FUNCTION_BLOCK TimeChannel1CH
VAR_INPUT
	EN: BOOL := TRUE;// Enable the time channel (settings must also be enabled)
	Speed            : INT;		// $(skip) 0,1=normal speed, 2=high speed
	OnTime           : UINT;	(* Hour/minute value of the switch-on time on the day *)
	OffTime          : UINT := 2400;	(* Hour/minute value of the switch-off time on the day *)
	Day: TimerDays;
	SingleShot       : BOOL;	(* $(skip) Resets EN after the on/off cycle is complete *)   
END_VAR
VAR_OUTPUT
	ENO: BOOL; // $(skip) Set if enabled and settings are valid
	Q: BOOL; // Result of the time channel
	Error: BOOL; // Settings error
	ErrorID: UDINT; // // $(skip) 1 = Inconsistent weekday settings, 2 = Bad time settings, 3 = on and off times equal
END_VAR
VAR
	CurrentDay: WORD; // $(skip)
	DayMatch: BOOL; // $(skip)
	LocalSystemTime: FB_LocalSystemTime; // $(skip)
	IsOnTime: BOOL; // $(skip)
	MinuteOfDay: WORD; // $(skip)
	StartMinuteOfDay: WORD; // $(skip)
	EndMinuteOfDay: WORD; // $(skip)
	Loop: WORD := 0; // $(skip)
	OnHour           : UINT;	(* $(skip) Hour value of the switch-on time on the day *)
	OnMinute         : UINT;	(* $(skip) Minute value of the switch-on time on the day *)
	OffHour          : UINT;	(* $(skip) Hour value of the switch-off time on the day *)
	OffMinute        : UINT;	(* $(skip) Minute value of the switch-off time on the day *)
END_VAR

Loop := Loop + 1;
Error := False;
IF Loop >= 10 THEN
	Loop := 0;
	OnHour := OnTime / 100;
	OnMinute := OnTime MOD 100;
	OffHour := OffTime / 100;
	OffMinute := OffTime MOD 100;
	LocalSystemTime(bEnable := TRUE);
	IF EN AND (NOT Error) THEN
		IF LocalSystemTime.bValid THEN	
			CurrentDay := F_GetDayOfWeek(in := NowDT()); 
			DayMatch := Day = TimerDays.AllDays OR (TO_WORD(Day) = CurrentDay - 1);
			IF OnHour = OffHour AND OnMinute = OffMinute THEN
				Q := FALSE;
			ELSE
				MinuteOfDay := LocalSystemTime.systemTime.wHour * 60 + LocalSystemTime.systemTime.wMinute;
				StartMinuteOfDay := OnHour * 60 + OnMinute;
				EndMinuteOfDay := OffHour * 60 + OffMinute;
				IsOnTime := MinuteOfDay >= StartMinuteOfDay AND MinuteOfDay < EndMinuteOfDay;
				Q := DayMatch AND IsOnTime;				
				IF Q AND SingleShot THEN
					EN := FALSE;
				END_IF
			END_IF
			ENO := TRUE;
		ELSE
			Q := FALSE;
			ENO := FALSE;
		END_IF
	ELSE
		Q := FALSE;
		ENO := FALSE;
	END_IF
END_IF

END_FUNCTION_BLOCK

(* stored: Version 1.1.0.1, ProductVersion 3.1.4024.6
   POU TimeChannel1CH: Id {817b1f2b-aa0c-4f9b-9e15-9571de197f24}, SpecialFunc None *)
